(* PLC project Unnamed, Unknown Unnamed 1 *)
(* stored: creationDateTime 2026-05-01T22:52:19, modificationDateTime 2026-05-02T15:13:44 *)

PROGRAM Project_04_Pneumatic_Pick_and_Place
  VAR
    PB_EStop AT %IX0.0 : BOOL;
    PB_Stop AT %IX0.1 : BOOL;
    PB_Start AT %IX0.2 : BOOL;
    PB_FaultReset AT %IX0.3 : BOOL;
    SW_ModeAuto AT %IX0.4 : BOOL;
    SEN_PartPresent AT %IX0.5 : BOOL;
    SEN_PartType AT %IX0.6 : BOOL;
    SEN_X_Home AT %IX0.7 : BOOL;
    SEN_X_Extended AT %IX1.0 : BOOL;
    SEN_Z_Up AT %IX1.1 : BOOL;
    SEN_Z_Down AT %IX1.2 : BOOL;
    SEN_Grip_Open AT %IX1.3 : BOOL;
    SEN_Grip_Closed AT %IX1.4 : BOOL;
    SEN_Reject_Home AT %IX1.5 : BOOL;
    SEN_Reject_Extended AT %IX1.6 : BOOL;
    SEN_TrayFull AT %IX1.7 : BOOL;
    SOL_X_Extend AT %QX0.0 : BOOL;
    SOL_X_Retract AT %QX0.1 : BOOL;
    SOL_Z_Down AT %QX0.2 : BOOL;
    SOL_Z_Up AT %QX0.3 : BOOL;
    SOL_Grip_Close AT %QX0.4 : BOOL;
    SOL_Grip_Open AT %QX0.5 : BOOL;
    SOL_Reject_Extend AT %QX0.6 : BOOL;
    HL1_RunLamp AT %QX0.7 : BOOL;
    HL2_StopLamp AT %QX1.0 : BOOL;
    HL3_AlarmLamp AT %QX1.1 : BOOL;
    HL4_AutoLamp AT %QX1.2 : BOOL;
    BZ1_CycleBeep AT %QX1.3 : BOOL;
    MR_MasterEnable AT %MX0.0 : BOOL;
    MR_CycleActive AT %MX0.1 : BOOL;
    MR_CycleStopReq AT %MX0.2 : BOOL;
    MR_FaultActive AT %MX0.3 : BOOL;
    MR_FaultTimeout AT %MX0.4 : BOOL;
    MR_FaultSensor AT %MX0.5 : BOOL;
    MR_FaultTrayFull AT %MX0.6 : BOOL;
    MR_AutoMode AT %MX0.7 : BOOL;
    MR_ManualMode AT %MX1.0 : BOOL;
    MR_PartIsGood AT %MX1.1 : BOOL;
    MR_PartIsReject AT %MX1.2 : BOOL;
    MR_HomePosition AT %MX1.3 : BOOL;
    MR_StepAdvance AT %MX1.4 : BOOL;
    MR_CycleBeepTrig AT %MX1.5 : BOOL;
  END_VAR
  VAR
    StepTimeoutTime : TIME := T#8s;
    GripDelayTime : TIME := T#300ms;
    PartDetectTime : TIME := T#500ms;
    RejectHoldTime : TIME := T#1s;
    BeepTime : TIME := T#200ms;
    CurrentStep : INT := 0;
    GoodPartsCount : INT := 0;
    RejectCount : INT := 0;
    CycleCount : INT := 0;
    FaultStep : INT := 0;
    PreviousStep : INT := 0;
    Zero : INT := 0;
    One : INT := 1;
    Two : INT := 2;
    Three : INT := 3;
    Four : INT := 4;
    Five : INT := 5;
    Six : INT := 6;
    Seven : INT := 7;
    eight : INT := 8;
    nine : INT := 9;
    Ten : INT := 10;
    II : INT := 11;
    I2 : INT := 12;
    I3 : INT := 13;
    I4 : INT := 14;
    I5 : INT := 15;
    TON_StepTimeout : TON;
    TON_PartDetectDly : TON;
    TON0 : TON;
    TON_GripDelay : TON;
    TON_RejectHold : TON;
    TON_BeepPulse : TON;
  END_VAR
  VAR  (* added by the conversion: wires and edge detectors of the diagram *)
    _EQ63_OUT : BOOL;
    _EQ172_OUT : BOOL;
    _EQ179_OUT : BOOL;
    _EQ197_ENO : BOOL;
    _EQ197_OUT : BOOL;
    _EQ198_ENO : BOOL;
    _EQ198_OUT : BOOL;
    _EQ206_ENO : BOOL;
    _EQ206_OUT : BOOL;
    _EQ207_ENO : BOOL;
    _EQ207_OUT : BOOL;
    _GE214_ENO : BOOL;
    _GE214_OUT : BOOL;
    _LE215_ENO : BOOL;
    _LE215_OUT : BOOL;
    _GE225_ENO : BOOL;
    _GE225_OUT : BOOL;
    _LE226_ENO : BOOL;
    _LE226_OUT : BOOL;
    _GE233_ENO : BOOL;
    _GE233_OUT : BOOL;
    _GE241_ENO : BOOL;
    _GE241_OUT : BOOL;
    _GE242_ENO : BOOL;
    _GE242_OUT : BOOL;
  END_VAR

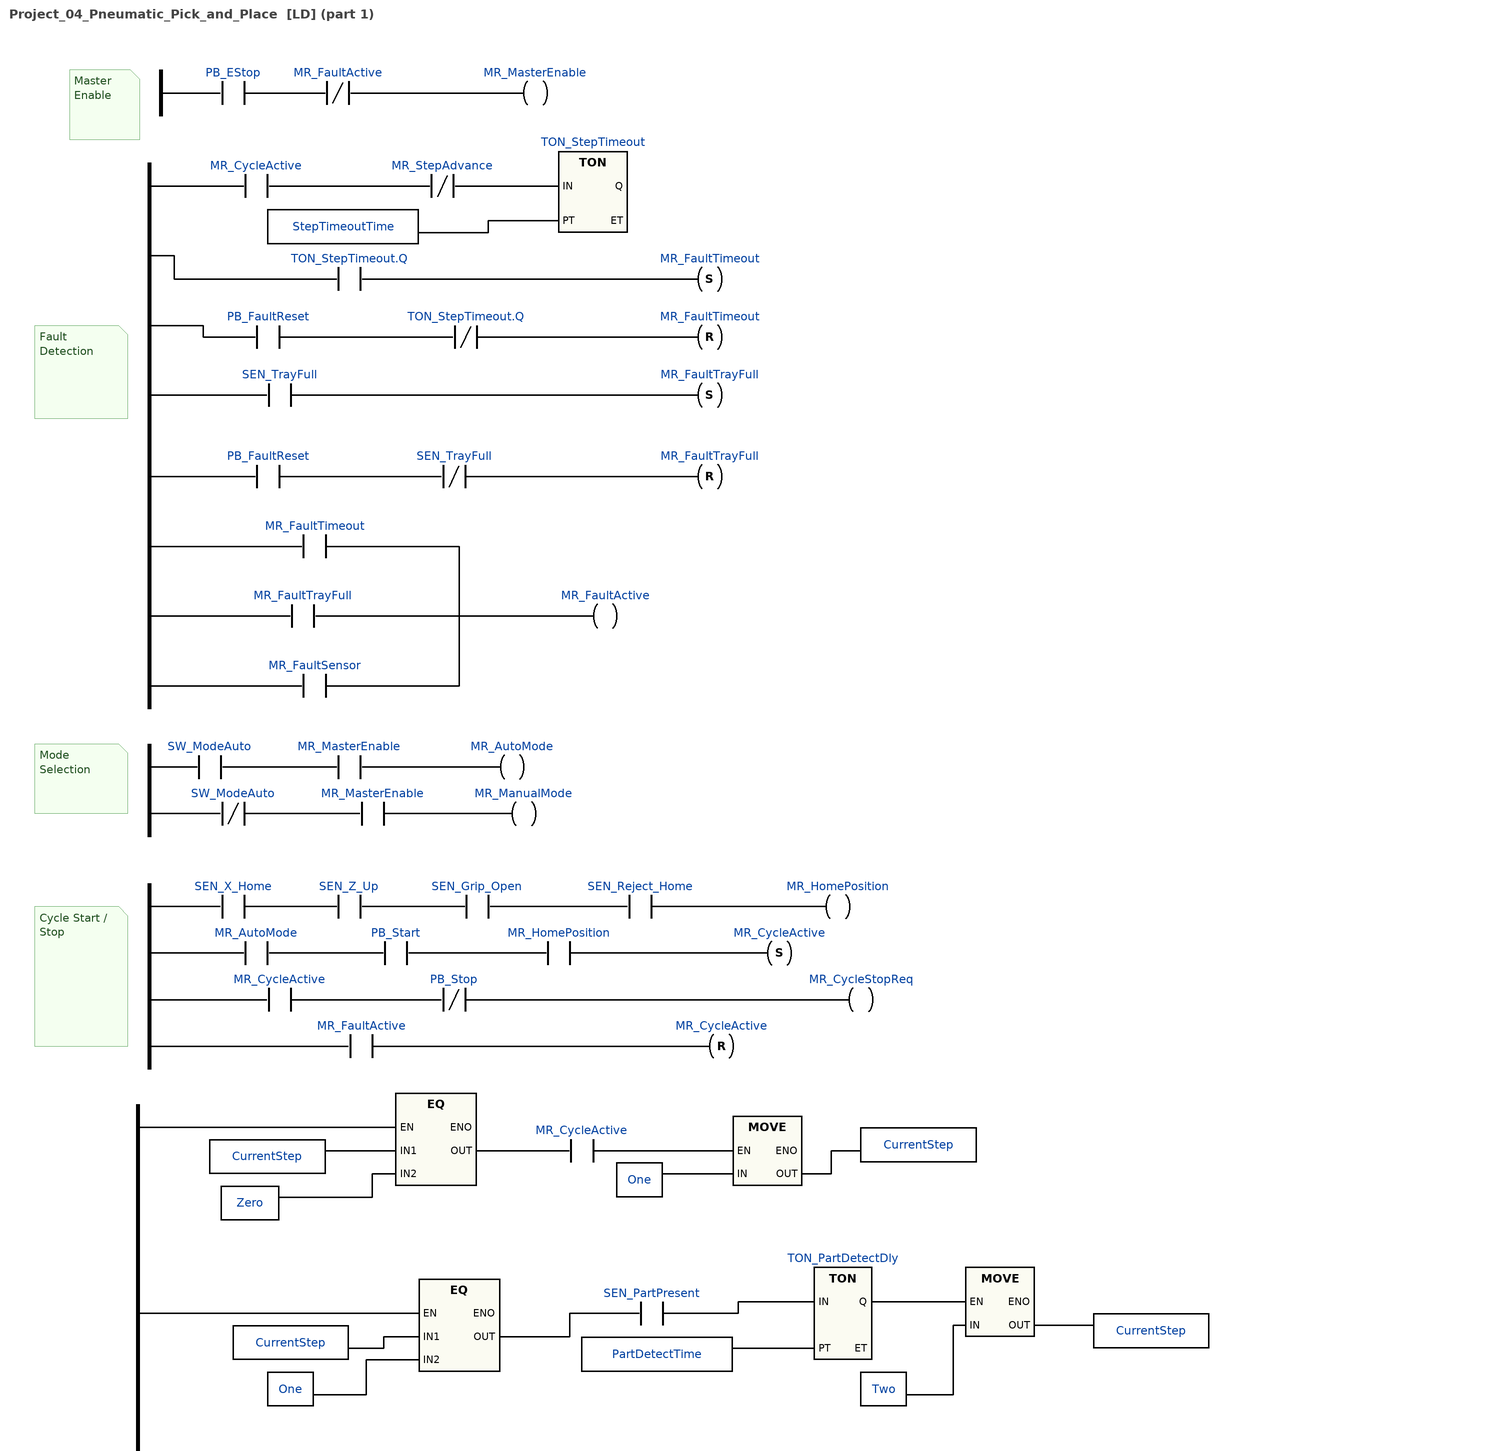
(* LD diagram, written out as Structured Text *)
(* Master Enable *)
MR_MasterEnable := PB_EStop AND NOT MR_FaultActive;
IF TON_StepTimeout.Q THEN MR_FaultTimeout := TRUE; END_IF;
(* Fault Detection *)
IF PB_FaultReset AND NOT TON_StepTimeout.Q THEN MR_FaultTimeout := FALSE; END_IF;
IF SEN_TrayFull THEN MR_FaultTrayFull := TRUE; END_IF;
IF PB_FaultReset AND NOT SEN_TrayFull THEN MR_FaultTrayFull := FALSE; END_IF;
MR_FaultActive := MR_FaultTrayFull OR MR_FaultTimeout OR MR_FaultSensor;
(* Mode Selection *)
MR_AutoMode := SW_ModeAuto AND MR_MasterEnable;
MR_ManualMode := NOT SW_ModeAuto AND MR_MasterEnable;
MR_HomePosition := SEN_X_Home AND SEN_Z_Up AND SEN_Grip_Open AND SEN_Reject_Home;
(* Cycle Start / Stop *)
IF MR_AutoMode AND PB_Start AND MR_HomePosition THEN MR_CycleActive := TRUE; END_IF;
MR_CycleStopReq := MR_CycleActive AND NOT PB_Stop;
IF MR_FaultActive THEN MR_CycleActive := FALSE; END_IF;
IF CurrentStep = Zero AND MR_CycleActive THEN CurrentStep := One; END_IF;
TON_PartDetectDly(IN := CurrentStep = One AND SEN_PartPresent, PT := PartDetectTime);
IF TON_PartDetectDly.Q THEN CurrentStep := Two; END_IF;
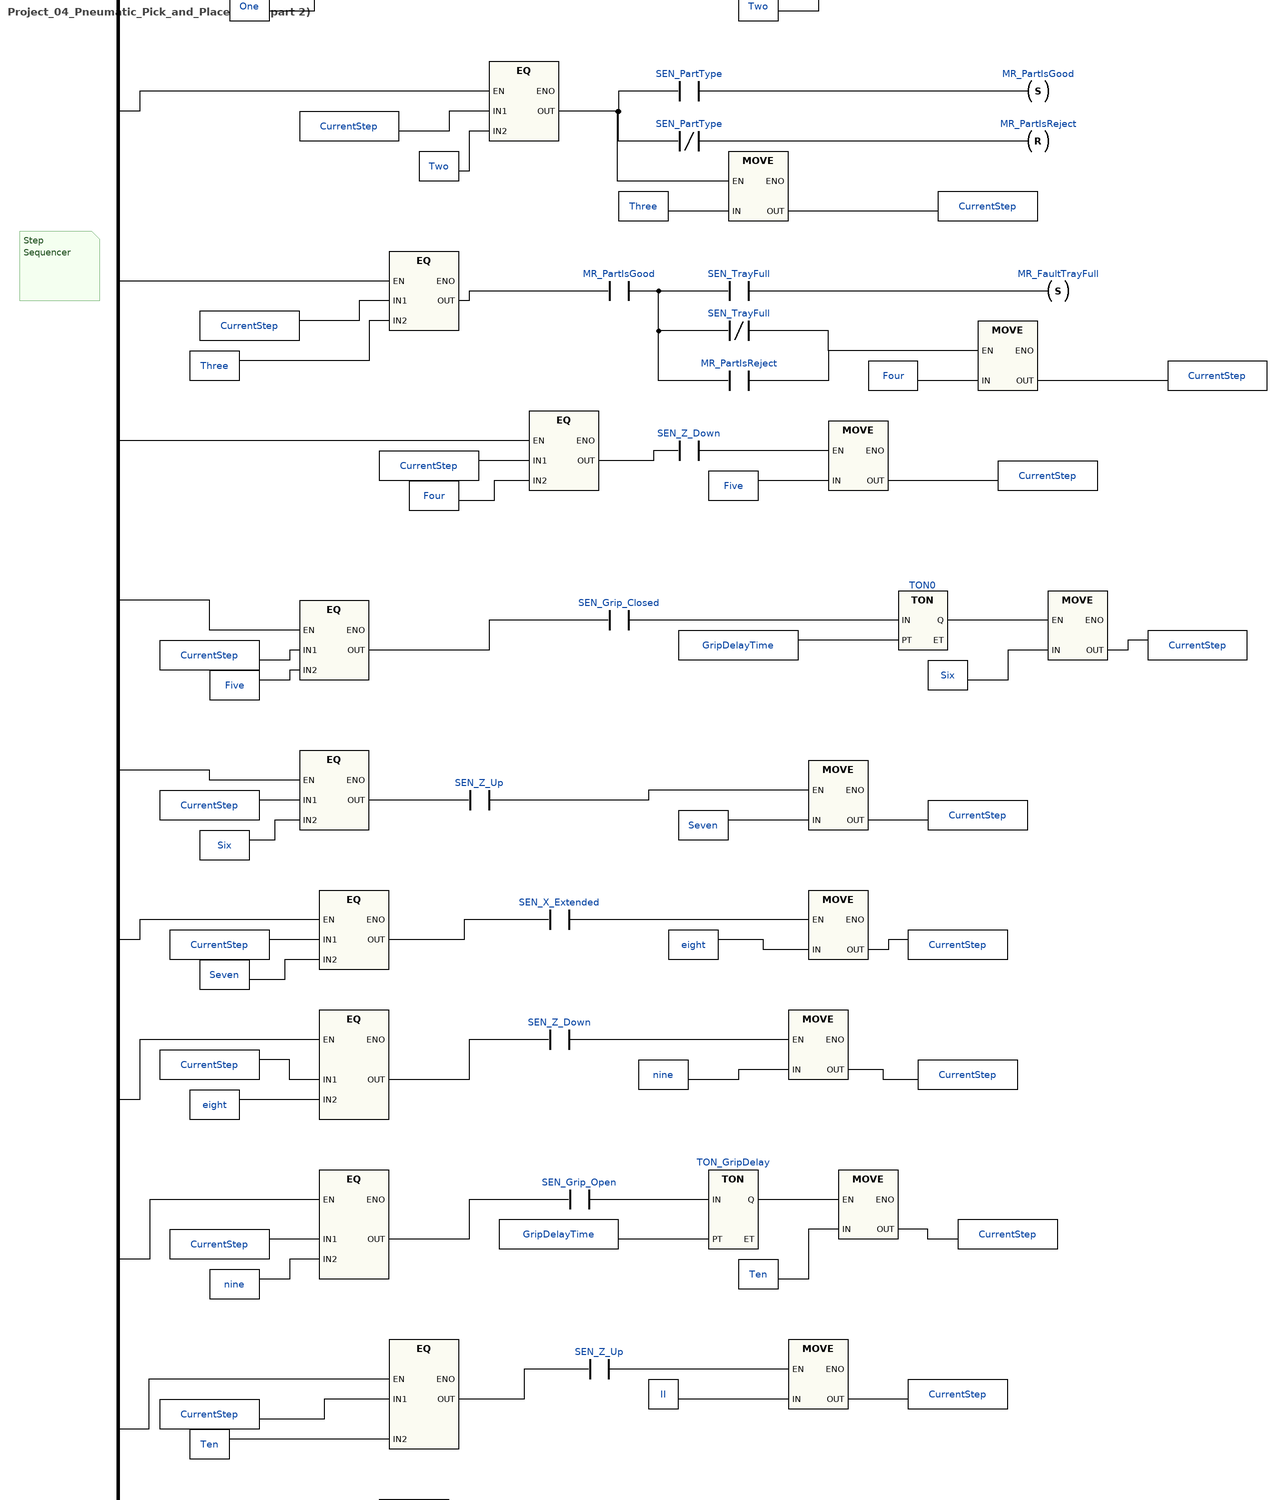
_EQ63_OUT := CurrentStep = Two;
IF _EQ63_OUT AND SEN_PartType THEN MR_PartIsGood := TRUE; END_IF;
IF _EQ63_OUT AND NOT SEN_PartType THEN MR_PartIsReject := FALSE; END_IF;
IF _EQ63_OUT THEN CurrentStep := Three; END_IF;
(* Step Sequencer *)
IF CurrentStep = Three AND MR_PartIsGood AND SEN_TrayFull THEN MR_FaultTrayFull := TRUE; END_IF;
IF CurrentStep = Three AND MR_PartIsGood AND (NOT SEN_TrayFull OR MR_PartIsReject) THEN CurrentStep := Four; END_IF;
IF CurrentStep = Four AND SEN_Z_Down THEN CurrentStep := Five; END_IF;
TON0(IN := CurrentStep = Five AND SEN_Grip_Closed, PT := GripDelayTime);
IF TON0.Q THEN CurrentStep := Six; END_IF;
IF CurrentStep = Six AND SEN_Z_Up THEN CurrentStep := Seven; END_IF;
IF CurrentStep = Seven AND SEN_X_Extended THEN CurrentStep := eight; END_IF;
IF CurrentStep = eight AND SEN_Z_Down THEN CurrentStep := nine; END_IF;
TON_GripDelay(IN := CurrentStep = nine AND SEN_Grip_Open, PT := GripDelayTime);
IF TON_GripDelay.Q THEN CurrentStep := Ten; END_IF;
IF CurrentStep = Ten AND SEN_Z_Up THEN CurrentStep := II; END_IF;
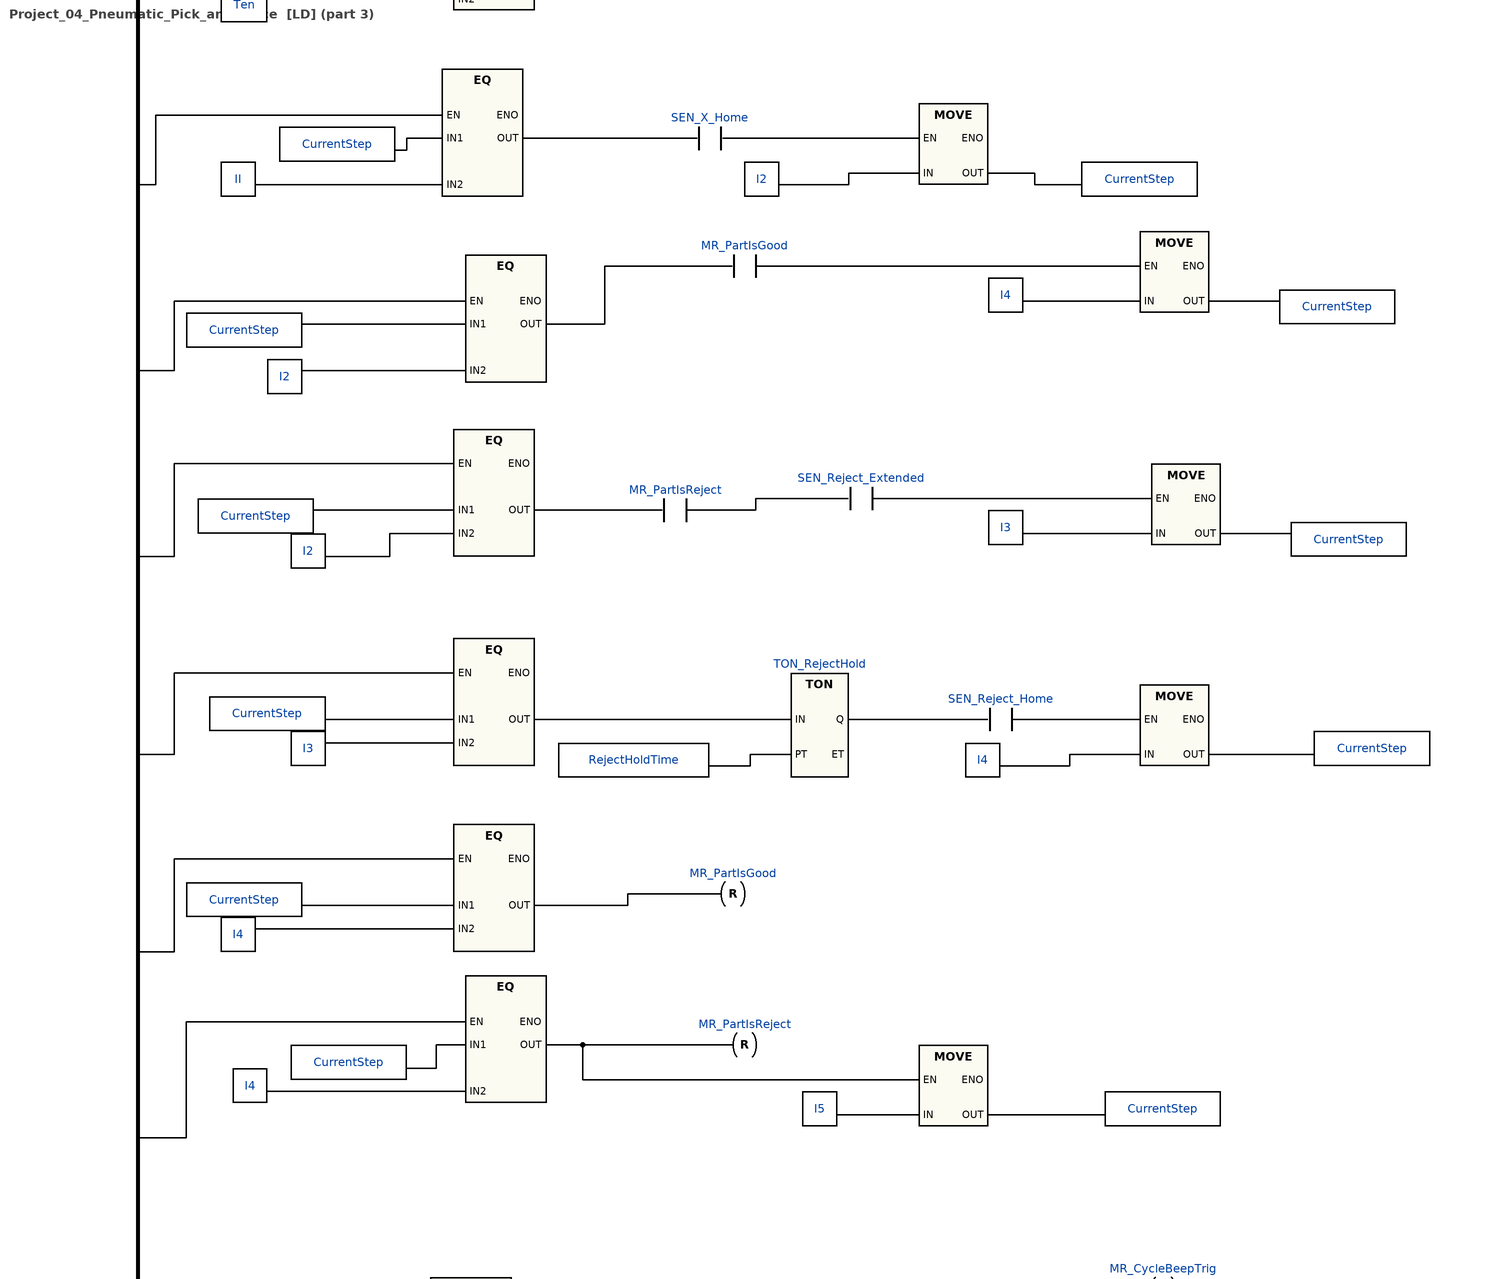
IF CurrentStep = II AND SEN_X_Home THEN CurrentStep := I2; END_IF;
IF CurrentStep = I2 AND MR_PartIsGood THEN CurrentStep := I4; END_IF;
IF CurrentStep = I2 AND MR_PartIsReject AND SEN_Reject_Extended THEN CurrentStep := I3; END_IF;
TON_RejectHold(IN := CurrentStep = I3, PT := RejectHoldTime);
IF TON_RejectHold.Q AND SEN_Reject_Home THEN CurrentStep := I4; END_IF;
IF CurrentStep = I4 THEN MR_PartIsGood := FALSE; END_IF;
_EQ172_OUT := CurrentStep = I4;
IF _EQ172_OUT THEN MR_PartIsReject := FALSE; END_IF;
IF _EQ172_OUT THEN CurrentStep := I5; END_IF;
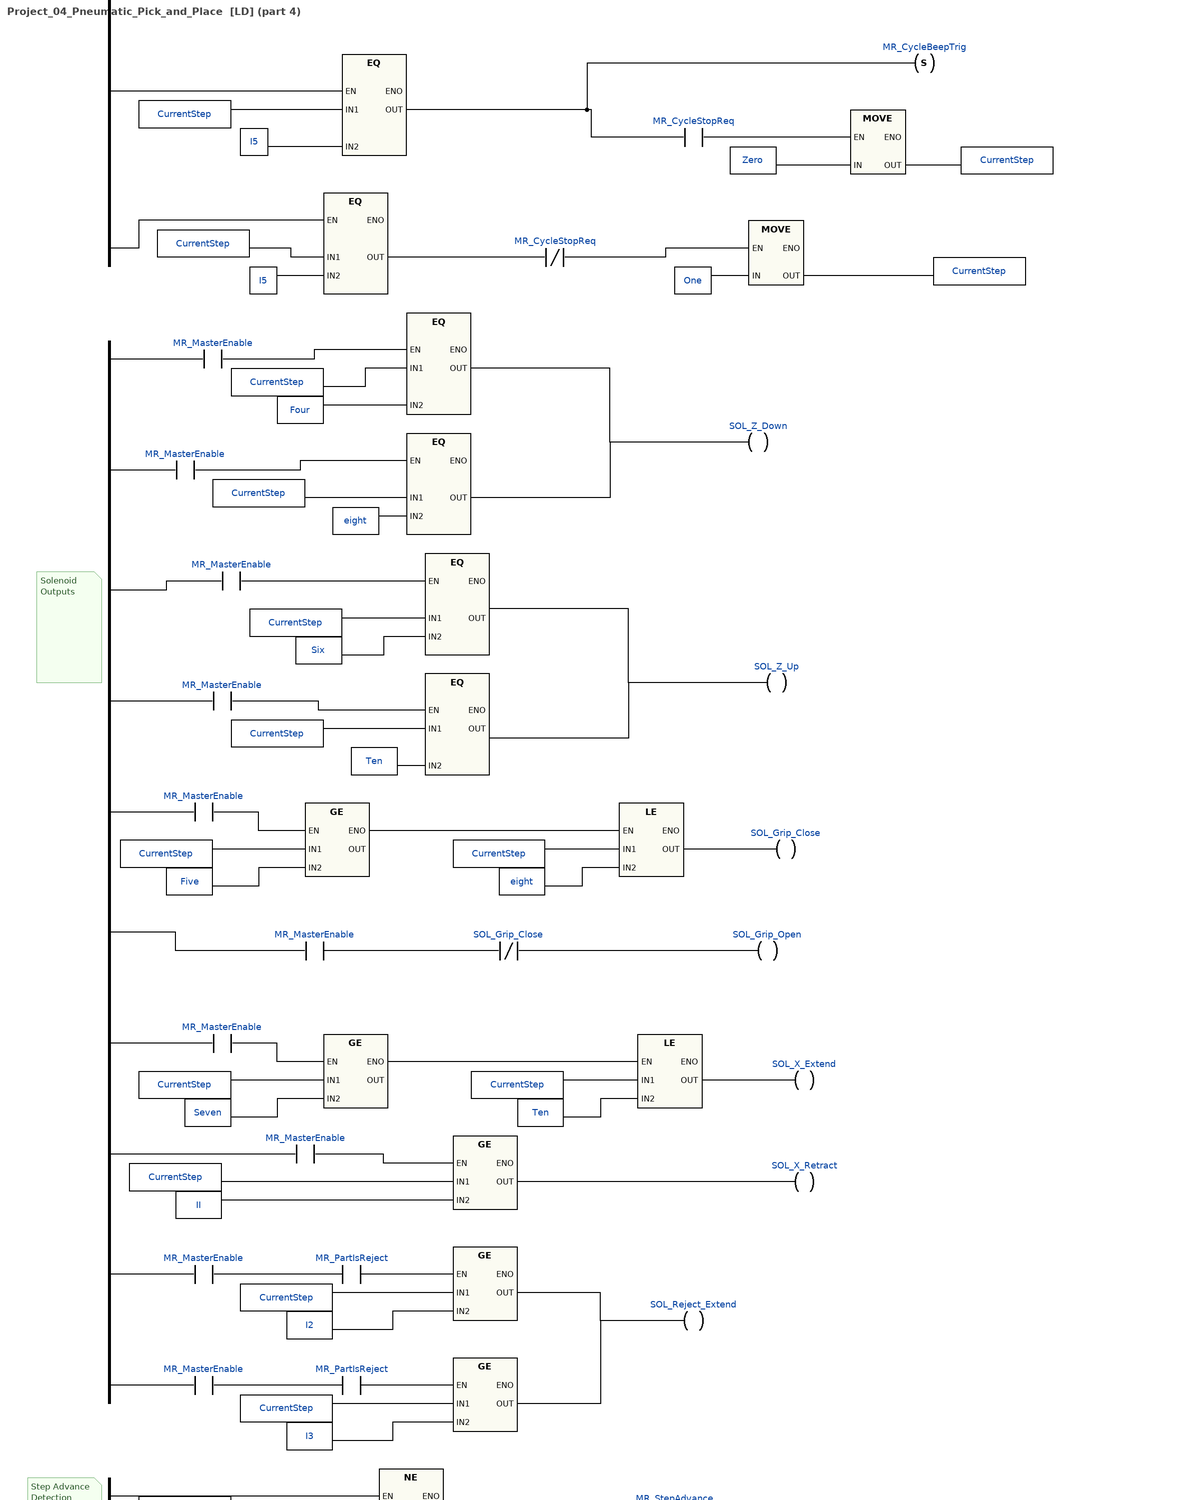
_EQ179_OUT := CurrentStep = I5;
IF _EQ179_OUT THEN MR_CycleBeepTrig := TRUE; END_IF;
IF _EQ179_OUT AND MR_CycleStopReq THEN CurrentStep := Zero; END_IF;
IF CurrentStep = I5 AND NOT MR_CycleStopReq THEN CurrentStep := One; END_IF;
_EQ197_OUT := EQ(EN := MR_MasterEnable, IN1 := CurrentStep, IN2 := Four, ENO => _EQ197_ENO);
_EQ198_OUT := EQ(EN := MR_MasterEnable, IN1 := CurrentStep, IN2 := eight, ENO => _EQ198_ENO);
SOL_Z_Down := _EQ197_OUT OR _EQ198_OUT;
(* Solenoid Outputs *)
_EQ206_OUT := EQ(EN := MR_MasterEnable, IN1 := CurrentStep, IN2 := Six, ENO => _EQ206_ENO);
_EQ207_OUT := EQ(EN := MR_MasterEnable, IN1 := CurrentStep, IN2 := Ten, ENO => _EQ207_ENO);
SOL_Z_Up := _EQ206_OUT OR _EQ207_OUT;
_GE214_OUT := GE(EN := MR_MasterEnable, IN1 := CurrentStep, IN2 := Five, ENO => _GE214_ENO);
_LE215_OUT := LE(EN := _GE214_ENO, IN1 := CurrentStep, IN2 := eight, ENO => _LE215_ENO);
SOL_Grip_Close := _LE215_OUT;
SOL_Grip_Open := MR_MasterEnable AND NOT SOL_Grip_Close;
_GE225_OUT := GE(EN := MR_MasterEnable, IN1 := CurrentStep, IN2 := Seven, ENO => _GE225_ENO);
_LE226_OUT := LE(EN := _GE225_ENO, IN1 := CurrentStep, IN2 := Ten, ENO => _LE226_ENO);
SOL_X_Extend := _LE226_OUT;
_GE233_OUT := GE(EN := MR_MasterEnable, IN1 := CurrentStep, IN2 := II, ENO => _GE233_ENO);
SOL_X_Retract := _GE233_OUT;
_GE241_OUT := GE(EN := MR_MasterEnable AND MR_PartIsReject, IN1 := CurrentStep, IN2 := I2, ENO => _GE241_ENO);
_GE242_OUT := GE(EN := MR_MasterEnable AND MR_PartIsReject, IN1 := CurrentStep, IN2 := I3, ENO => _GE242_ENO);
SOL_Reject_Extend := _GE241_OUT OR _GE242_OUT;
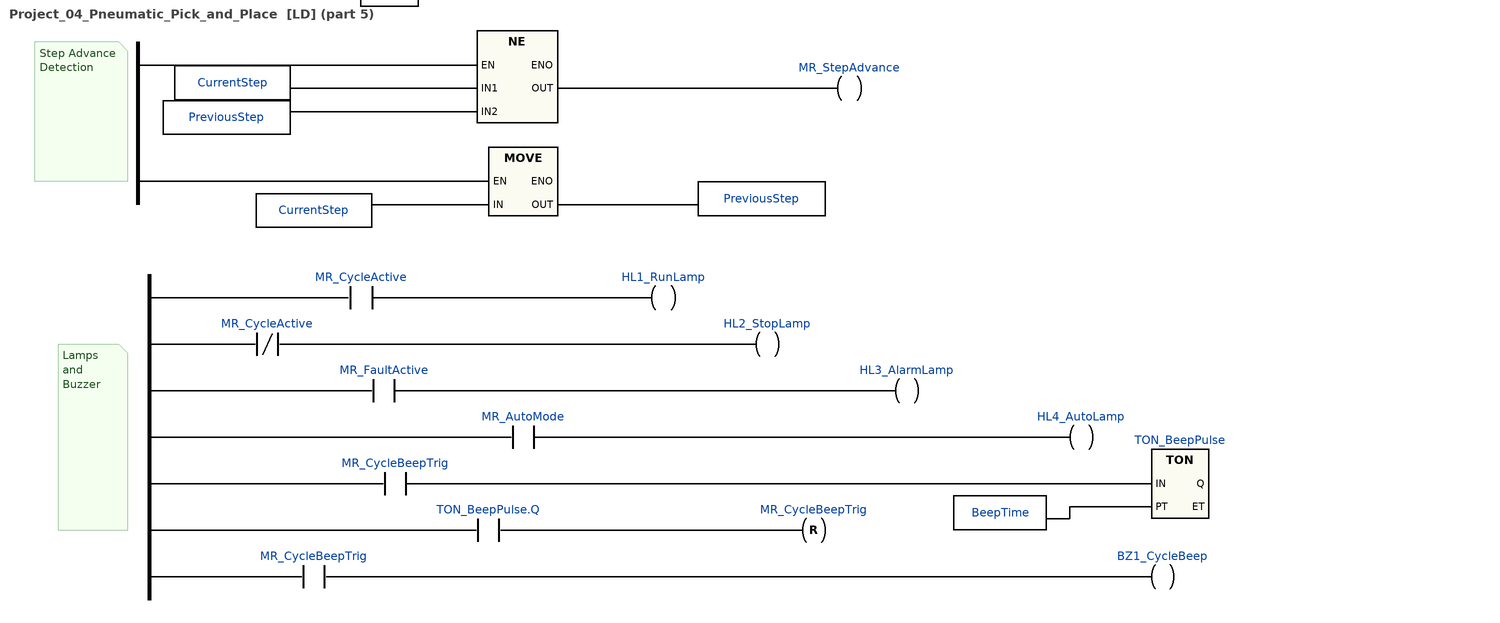
(* Step Advance Detection *)
MR_StepAdvance := CurrentStep <> PreviousStep;
PreviousStep := CurrentStep;
HL1_RunLamp := MR_CycleActive;
HL2_StopLamp := NOT MR_CycleActive;
(* Lamps and Buzzer *)
HL3_AlarmLamp := MR_FaultActive;
HL4_AutoLamp := MR_AutoMode;
IF TON_BeepPulse.Q THEN MR_CycleBeepTrig := FALSE; END_IF;
BZ1_CycleBeep := MR_CycleBeepTrig;
TON_StepTimeout(IN := MR_CycleActive AND NOT MR_StepAdvance, PT := StepTimeoutTime);
TON_BeepPulse(IN := MR_CycleBeepTrig, PT := BeepTime);
END_PROGRAM

CONFIGURATION Config0
  RESOURCE Res0 ON PLC
    TASK task0(INTERVAL := T#20ms, PRIORITY := 0);
    PROGRAM instance0 WITH task0 : Project_04_Pneumatic_Pick_and_Place;
  END_RESOURCE
END_CONFIGURATION
